(* PLC project Blank Project, Blank Blank 1.0 *)
(* stored: creationDateTime 2016-05-18T21:14:07, modificationDateTime 2017-10-17T19:47:22 *)

PROGRAM Cell3
  VAR
    C2_IR AT %IX0.3 : BOOL := true;
    M2_IR AT %IX0.4 : BOOL := true;
    Main AT %IX0.6 : BOOL := true;
    M2_motor AT %QX0.2 : BOOL := true;
    C3_motor AT %QX0.4 : BOOL := true;
  END_VAR
  VAR
    C3_working : BOOL := false;
  END_VAR
  VAR
    C3_working_int AT %MD1 : DINT := 0;
  END_VAR
  VAR
    C3_afterM : BOOL := false;
  END_VAR
  VAR
    C3_afterM_int AT %MD2 : DINT := 0;
  END_VAR
  VAR
    Step1 : BOOL := false;
  END_VAR
  VAR
    Step1_int AT %MD3 : DINT := 0;
  END_VAR
  VAR
    Step2 : BOOL := false;
  END_VAR
  VAR
    Step2_int AT %MD4 : DINT := 0;
  END_VAR
  VAR
    Pause : BOOL := false;
  END_VAR
  VAR
    Pause_int AT %MD5 : DINT := 0;
  END_VAR
  VAR
    Timer_conveyor : TON;
    Timer_machining : TON;
    TON1 : TON;
    TON2 : TON;
    TON3 : TON;
  END_VAR
  VAR
    JadeProg1 AT %IX0.7 : BOOL := true;
  END_VAR
  VAR
    TON0 : TON;
  END_VAR

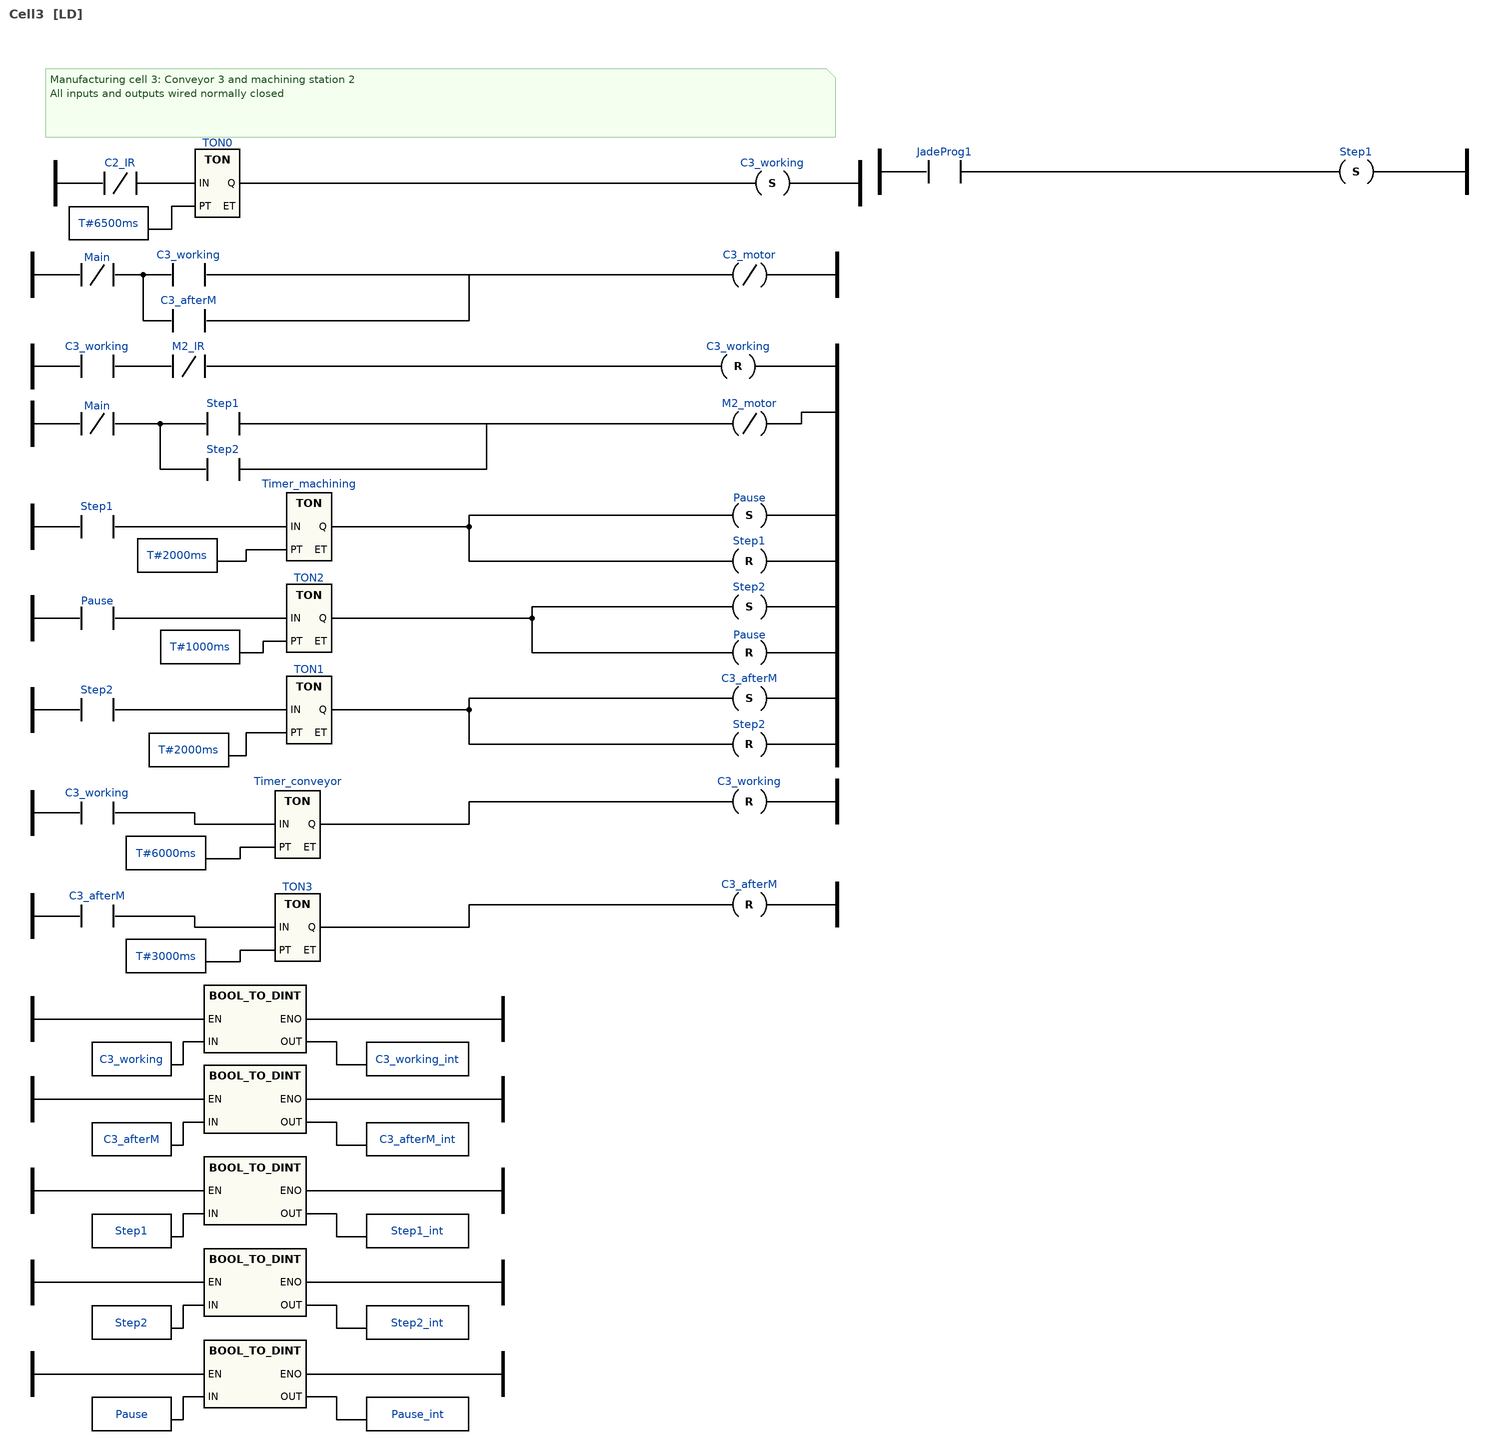
(* LD diagram, written out as Structured Text *)
(* Manufacturing cell 3: Conveyor 3 and machining station 2
All inputs and outputs wired normally closed *)
IF JadeProg1 THEN Step1 := TRUE; END_IF;
TON0(IN := NOT C2_IR, PT := T#6500ms);
IF TON0.Q THEN C3_working := TRUE; END_IF;
C3_motor := NOT (NOT Main AND (C3_working OR C3_afterM));
IF C3_working AND NOT M2_IR THEN C3_working := FALSE; END_IF;
M2_motor := NOT (NOT Main AND (Step1 OR Step2));
Timer_machining(IN := Step1, PT := T#2000ms);
IF Timer_machining.Q THEN Pause := TRUE; END_IF;
IF Timer_machining.Q THEN Step1 := FALSE; END_IF;
TON2(IN := Pause, PT := T#1000ms);
IF TON2.Q THEN Step2 := TRUE; END_IF;
IF TON2.Q THEN Pause := FALSE; END_IF;
TON1(IN := Step2, PT := T#2000ms);
IF TON1.Q THEN C3_afterM := TRUE; END_IF;
IF TON1.Q THEN Step2 := FALSE; END_IF;
Timer_conveyor(IN := C3_working, PT := T#6000ms);
IF Timer_conveyor.Q THEN C3_working := FALSE; END_IF;
TON3(IN := C3_afterM, PT := T#3000ms);
IF TON3.Q THEN C3_afterM := FALSE; END_IF;
C3_working_int := BOOL_TO_DINT(C3_working);
C3_afterM_int := BOOL_TO_DINT(C3_afterM);
Step1_int := BOOL_TO_DINT(Step1);
Step2_int := BOOL_TO_DINT(Step2);
Pause_int := BOOL_TO_DINT(Pause);
END_PROGRAM

CONFIGURATION Config0
  RESOURCE Res0 ON PLC
    TASK TaskMain(INTERVAL := T#50ms, PRIORITY := 0);
    PROGRAM Inst0 WITH TaskMain : Cell3;
  END_RESOURCE
END_CONFIGURATION
